FUNCTION_BLOCK NeredaCapacitySpToCBlowersSp (* Basic Function Block Type *)
  (* Standard: 61499-2 *)
  (* Version 1.0, 9/29/2026, SESA685388, Schneider Electric, Rev1 - MaxSp sempre forca 100% (inclusive nas fases C2/C3) *)
  PACKAGE SE.Nereda;
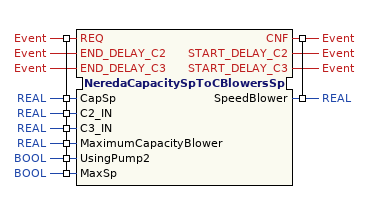
  EVENT_INPUT
    REQ WITH CapSp, C2_IN, C3_IN, UsingPump2, MaximumCapacityBlower, MaxSp;
    END_DELAY_C2;
    END_DELAY_C3;
  END_EVENT
  EVENT_OUTPUT
    CNF WITH SpeedBlower; (* Execution Confirmation *)
    START_DELAY_C2;
    START_DELAY_C3;
  END_EVENT
  VAR_INPUT
    CapSp : REAL; (* Input event qualifier *)
    C2_IN : REAL;
    C3_IN : REAL;
    MaximumCapacityBlower : REAL;
    UsingPump2 : BOOL;
    MaxSp : BOOL;
  END_VAR
  VAR_OUTPUT
    SpeedBlower : REAL;
  END_VAR
  VAR
    LastUsingPump2 : BOOL;
    Starting2Pumps : BOOL;
    Stopping1Pump : BOOL;
  END_VAR
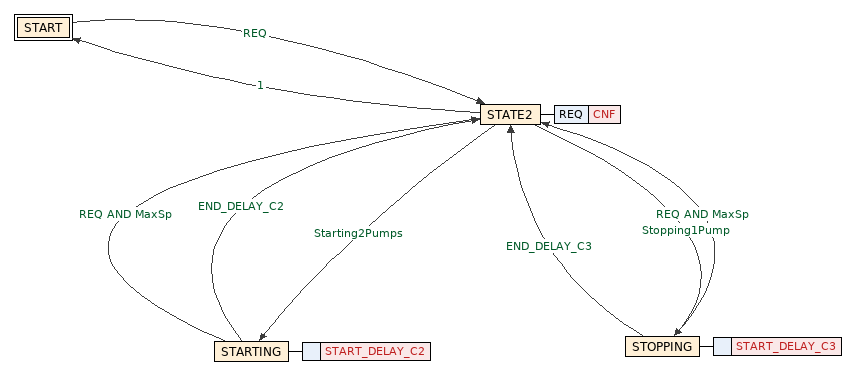
  EC_STATES
    START; (* Initial State *)
    STATE2 : REQ -> CNF;
    STARTING : -> START_DELAY_C2;
    STOPPING : -> START_DELAY_C3;
  END_STATES
  EC_TRANSITIONS
    START TO STATE2 := REQ;
    STATE2 TO STARTING := Starting2Pumps;
    STARTING TO STATE2 := END_DELAY_C2;
    STATE2 TO STOPPING := Stopping1Pump;
    STOPPING TO STATE2 := END_DELAY_C3;
    STARTING TO STATE2 := REQ AND MaxSp;
    STOPPING TO STATE2 := REQ AND MaxSp;
    STATE2 TO START := 1;
  END_TRANSITIONS
  ALGORITHM REQ IN ST: (* Initialization algorithm *)
;
IF (UsingPump2 AND NOT(LastUsingPump2)) THEN
	Starting2Pumps:=TRUE;
ELSE
	Starting2Pumps:=FALSE;
END_IF;

IF (NOT UsingPump2 AND LastUsingPump2) THEN
	Stopping1Pump := TRUE;
ELSE
	Stopping1Pump := FALSE;
END_IF;


IF (NOT UsingPump2 )THEN
    // Zone 1 : 0 ... C2_IN  =>  0 ... 100 %
    IF Stopping1Pump THEN
	    SpeedBlower := C3_IN;
    ELSE
    	SpeedBlower := MIN((CapSp / MaximumCapacityBlower) * 100.0, 100);
    END_IF;
END_IF;

IF (UsingPump2 )THEN
    // Zone 1 : 0 ... C2_IN  =>  0 ... 100 %
    IF Starting2Pumps THEN
	    SpeedBlower := C2_IN;
    ELSE
    	SpeedBlower := (CapSp / (2*MaximumCapacityBlower)) * 100.0;
    END_IF;
END_IF;

// Rev1: reator acima de Cmax com 1 soprador soprando de fato (MaxSp) fica
// SEMPRE no maximo, inclusive na saida de um soprador (fase C3).
IF MaxSp THEN
	SpeedBlower := 100.0;
END_IF;

LastUsingPump2:=UsingPump2;
  END_ALGORITHM
END_FUNCTION_BLOCK
